// TIA Portal V20 export
TYPE "UDT_MaintenanceTask"
   STRUCT
      Elapsed : Bool;
      Id : Bool;
      Period : Bool;
      Warning : Bool;
   END_STRUCT;
END_TYPE
